// TIA Portal V16 export
// export: Created 2021-04-11T09:51:32.9894419Z, ExportSetting WithDefaults, DisplayName Totally Integrated Automation Portal, DisplayVersion V16, DisplayName TIA Portal Version Control Interface, DisplayVersion V16, DisplayName TIA Portal Openness, DisplayVersion V16, DisplayName STEP 7 Professional, DisplayVersion V16, DisplayName STEP 7 Safety, DisplayVersion V16, DisplayName WinCC Unified SCADA Engineering System, DisplayVersion V16
DATA_BLOCK "tst_DB"   // DB6
VERSION : 0.1
// stored: AutoNumber true, DBAccessibleFromOPCUA true, InstanceOfName tst, InstanceOfType FB
"tst"
   // VAR
   //    abcDec : DInt;
   //    arrBin : Array[1..12] of Bool;
   //    qwer : Array[0..12] of Real;
   //    Sort_Real_Instance { S7_SetPoint := 'True'} : "Sort_Real";
   // END_VAR
BEGIN
END_DATA_BLOCK
